{attribute 'qualified_only'}
{attribute 'strict'}
TYPE MotionFunctions :
(
	MoveAbsolute	:= 0,
	MoveRelative	:=1,
	Jog				:=2,
	MoveVelocity	:=3,
	MoveModulo		:=4,
	SingleGearIn	:=5,
	SingleGearOut	:=6,
	MultiGear		:=7,
	Home			:=10
);
END_TYPE

(* stored: Version 1.1.0.1, ProductVersion 3.1.4022.10
   DUT MotionFunctions: Id {7dfb6efd-1034-45c3-ba43-5dc10decbfbc} *)
